# B&R Automation Studio project URTC-with-integrated-CNC-system-main
Automation Studio 4.5.2.102

## Configuration Real

CPU 4PP065.0571-P74, AutomationRuntime D4.52, Build 4.1.2, Vc V4.25.0, Safety 1.6

### Task classes (Cpu.sw)
```
Cyclic#1 (cycle 2000 us, tolerance 0 us):
  ncsdcctrl <- ncsdcctrl.prg
  SDCAxisCtr <- SDCAxisCtr.prg
  SDCAxisCt1 <- SDCAxisCtr1.prg
  SDCAxisCt2 <- SDCAxisCtr2.prg
DataObjects: Arnc0sys
NcDataObjects: AxisInit <- AxisInit.dob, gAxis03a <- gAxis03obj.gAxis03a.dob, gAxis03i <- gAxis03obj.gAxis03i.dob, AxisApt <- AxisApt.dob, gmcipvar <- GmcIpUserConfig.gmcipvar.dob, gmcipfun <- GmcIpUserConfig.gmcipfun.dob, gmcipfub <- GmcIpUserConfig.gmcipfub.dob, gmcipubr <- GmcIpUserConfig.gmcipubr.dob, gmcipusm <- GmcIpUserConfig.gmcipusm.dob, gmcipui <- GmcIpUserConfig.gmcipui.dob, gmcipus <- GmcIpUserConfig.gmcipus.dob, gmcipuc <- GmcIpUserConfig.gmcipuc.dob, gmcipsys <- GmcIpConfig.gmcipsys.dob, gmciplbr <- GmcIpConfig.gmciplbr.dob, gmcipcbr <- GmcIpConfig.gmcipcbr.dob, gmciplsm <- GmcIpConfig.gmciplsm.dob, gmcipcsm <- GmcIpConfig.gmcipcsm.dob, gmcipcfg <- GmcIpConfig.gmcipcfg.dob, gmcipiec <- GmcIpConfig.gmcipiec.dob, gmciplog <- GmcIpConfig.gmciplog.dob, gmcipesm <- GmcIpConfig.gmcipesm.dob, gmcipmxd <- GmcIpConfig.gmcipmxd.dob, gmcipmx <- GmcIpConfig.gmcipmx.dob, CncInit <- CncInit.dob, CncProg <- CncProg.dob, CncProg1 <- CncProg1.dob, gAxis04a <- gAxis04obj.gAxis04a.dob, gAxis04i <- gAxis04obj.gAxis04i.dob
Binaries: TCData, Acp10map1, acp10cfg, Acp10map, arconfig, User, Role, sysconf, iomap, asfw, ashwd, arnc0cfg, Arnc0map
Libraries: Acp10sdc, Library, Acp10man, Acp10_MC, sys_lib, brsystem, asstring, powerlnk, asieccon, AsMath, Arnc0man, DataObj, AsArLog, FileIO, AsArProf, AsMem, Runtime, astime, Acp10par, NcGlobal, asiotime, AsBrStr
```

### Hardware
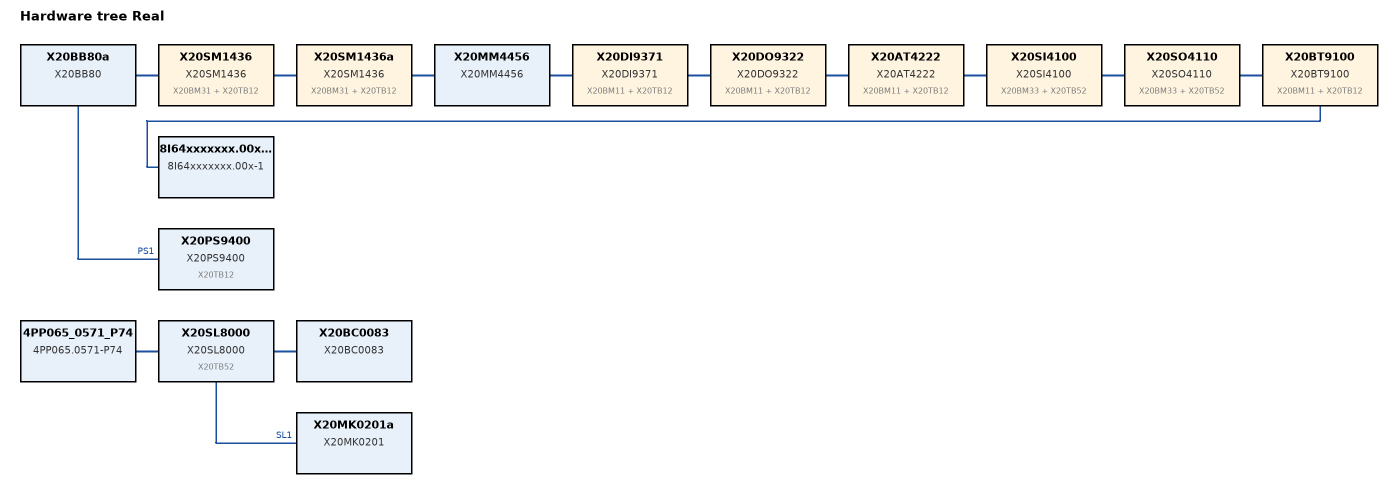
```
4PP065_0571_P74 : 4PP065.0571-P74 v1.1.2.0
  Connector IF4:
    EplInterfaceRedundant = 0
    EplEthInterfaceRedundant = 0
  Connector IF5:
    ActivateDevice = 1
    Mode = Manual
    InternetAddress = 10.0.1.10
    SubnetMask = 255.255.255.0
  ConfigurationID = labBR
  TimerDeviceType = EPLX2X
  TimerDevice = 4PP065_0571_P74.IF4
  TaskClassIdleTime = 2000
  Cyclic1Duration = 2000
  Cyclic1Tolerance = 0
  Cyclic1Output = 1
  Cyclic3Tolerance = 0
  VcObjectName = Visu
8I64xxxxxxx.00x-1 : 8I64xxxxxxx.00x-1 v2.1.2.0  [X2X1 -> X20BT9100.X2X1 [Cable Type=X2XCable, Length=10, Version=1.0.0.2]]
  BothEndSwitchesAreNormallyOpen_r1 = on
  QuickStopIsNormallyOpen_r1 = on
X20AT4222 : X20AT4222 v1.2.3.0  [SS1 -> X20TB12f.SS; SL -> X20BM11c.SL1]
X20BB80a : X20BB80 v1.0.2.0
X20BC0083 : X20BC0083 v2.9.0.0  [PLK1 -> X20SL8000.PLK2 (NodeNumber=2) [Cable Type=PowerlinkCable, Length=10, Version=1.0.0.2]; SL -> X20BB80a.SL1]
X20BM11a : X20BM11 v1.0.0.1  [X2X1 -> X20MM4456.X2X2]
X20BM11b : X20BM11 v1.0.0.1  [X2X1 -> X20BM11a.X2X2]
X20BM11c : X20BM11 v1.0.0.1  [X2X1 -> X20BM11b.X2X2]
X20BM11d : X20BM11 v1.0.0.1  [X2X1 -> X20BM33b.X2X2]
X20BM31a : X20BM31 v1.0.0.1  [X2X1 -> X20BB80a.IF1]
X20BM31b : X20BM31 v1.0.0.1  [X2X1 -> X20BM31a.X2X2]
X20BM33a : X20BM33 v1.0.0.4  [X2X1 -> X20BM11c.X2X2]
X20BM33b : X20BM33 v1.0.0.4  [X2X1 -> X20BM33a.X2X2]
X20BT9100 : X20BT9100 v1.0.3.0  [SS1 -> X20TB12g.SS; SL -> X20BM11d.SL1]
X20DI9371 : X20DI9371 v1.0.2.0  [SS1 -> X20TB12d.SS; SL -> X20BM11a.SL1]
X20DO9322 : X20DO9322 v1.0.3.0  [SS1 -> X20TB12e.SS; SL -> X20BM11b.SL1]
X20MK0201a : X20MK0201 v1.0.0.0  [SL -> X20SL8000.SL1]
X20MM4456 : X20MM4456 v1.1.5.0  [X2X1 -> X20BM31b.X2X2]
X20PS9400 : X20PS9400 v1.0.2.4  [SS1 -> X20TB12b.SS; PS -> X20BB80a.PS1]
X20SI4100 : X20SI4100 v1.10.1.1  [SS1 -> X20TB52b.SS; SL -> X20BM33a.SL1]
X20SL8000 : X20SL8000 v1.6.5.1  [PLK1 -> 4PP065_0571_P74.IF4 (NodeNumber=1) [Cable Type=PowerlinkCable, Length=10, Version=1.0.0.2]; PLK2 -> X20BC0083.PLK1 (NodeNumber=1) [Cable Type=PowerlinkCable, Length=10, Version=1.0.0.2]; SS1 -> X20TB52a.SS]
  SafeProject = SafeLOGIC-1
X20SM1436 : X20SM1436 v1.4.2.1  [SS1 -> X20TB12a.SS; SL -> X20BM31a.SL1]
X20SM1436a : X20SM1436 v1.4.2.1  [SS1 -> X20TB12c.SS; SL -> X20BM31b.SL1]
X20SO4110 : X20SO4110 v1.10.1.1  [SS1 -> X20TB52c.SS; SL -> X20BM33b.SL1]
  SafeLogicID = 2
  SafeModuleID = 3
X20TB12a : X20TB12 v1.0.0.0
X20TB12b : X20TB12 v1.0.0.0
X20TB12c : X20TB12 v1.0.0.0
X20TB12d : X20TB12 v1.0.0.0
X20TB12e : X20TB12 v1.0.0.0
X20TB12f : X20TB12 v1.0.0.0
X20TB12g : X20TB12 v1.0.0.0
X20TB52a : X20TB52 v1.0.0.1
X20TB52b : X20TB52 v1.0.0.1
X20TB52c : X20TB52 v1.0.0.1
```

### Acp10map.ncm - 4PP065_0571_P74/Motion/Acp10map.ncm
```
NcMapping (NcSwId=Acp10, DisabledNodesAreHidden=False)
  NcObject gAxis03 (ModuleId=8I64xxxxxxx.00x-1, ModuleAddress=SDC_IF1.ST1, Type=ncAXIS, Channel=1, AcoposSimulation=Off, InitParameter=gAxis03i, AcoposParameter=gAxis03a, AdditionalData=CNC_Enabled="1" , Disabled=FALSE, ModuleDisabled=FALSE)
```

### Acp10map1.ncm - 4PP065_0571_P74/Motion/Acp10map1.ncm
```
NcMapping (NcSwId=ACP10, DisabledNodesAreHidden=False)
  NcObject AxisX (ModuleAddress=SDC_IF1.ST2, InterfaceType=SDC, Type=ncAXIS, Channel=1, AcoposSimulation=Off, InitParameter=AxisInit, AcoposParameter=AxisApt, AdditionalData=CNC_Enabled="1" , Disabled=FALSE, ModuleDisabled=FALSE)
  NcObject AxisY (ModuleAddress=SDC_IF1.ST3, InterfaceType=SDC, Type=ncAXIS, Channel=1, AcoposSimulation=Off, InitParameter=AxisInit, AcoposParameter=AxisApt, AdditionalData=CNC_Enabled="1" , Disabled=FALSE)
  NcObject AxisZ (ModuleAddress=SDC_IF1.ST4, InterfaceType=SDC, Type=ncAXIS, Channel=1, AcoposSimulation=Off, InitParameter=AxisInit, AcoposParameter=AxisApt, AdditionalData=CNC_Enabled="1" , Disabled=FALSE)
```

### Arnc0map.ncm - 4PP065_0571_P74/Motion/Arnc0map.ncm
```
NcMapping (NcSwId=Arnc0, DisabledNodesAreHidden=False)
  NcObject CNCsys (Type=ncCNCSYS, Channel=1, AcoposSimulation=Off, InitParameter=CncInit, Disabled=FALSE, ModuleDisabled=FALSE)
  NcObject CNC2 (Type=ncCNCSYS, Channel=2, AcoposSimulation=Off, Disabled=TRUE, ModuleDisabled=FALSE)
  NcObject CNC3 (Type=ncCNCSYS, Channel=3, AcoposSimulation=Off, Disabled=TRUE, ModuleDisabled=FALSE)
  NcObject CNC4 (Type=ncCNCSYS, Channel=4, AcoposSimulation=Off, Disabled=TRUE, ModuleDisabled=FALSE)
  NcObject CNC5 (Type=ncCNCSYS, Channel=5, AcoposSimulation=Off, Disabled=TRUE, ModuleDisabled=FALSE)
  NcObject CNC6 (Type=ncCNCSYS, Channel=6, AcoposSimulation=Off, Disabled=TRUE, ModuleDisabled=FALSE)
  NcObject CNC7 (Type=ncCNCSYS, Channel=7, AcoposSimulation=Off, Disabled=TRUE, ModuleDisabled=FALSE)
  NcObject CNC8 (Type=ncCNCSYS, Channel=8, AcoposSimulation=Off, Disabled=TRUE, ModuleDisabled=FALSE)
  NcObject CNC9 (Type=ncCNCSYS, Channel=9, AcoposSimulation=Off, Disabled=TRUE, ModuleDisabled=FALSE)
  NcObject CNC10 (Type=ncCNCSYS, Channel=10, AcoposSimulation=Off, Disabled=TRUE, ModuleDisabled=FALSE)
  NcObject CNC11 (Type=ncCNCSYS, Channel=11, AcoposSimulation=Off, Disabled=TRUE, ModuleDisabled=FALSE)
  NcObject CNC12 (Type=ncCNCSYS, Channel=12, AcoposSimulation=Off, Disabled=TRUE, ModuleDisabled=FALSE)
  NcObject CNC13 (Type=ncCNCSYS, Channel=13, AcoposSimulation=Off, Disabled=TRUE, ModuleDisabled=FALSE)
  NcObject CNC14 (Type=ncCNCSYS, Channel=14, AcoposSimulation=Off, Disabled=TRUE, ModuleDisabled=FALSE)
  NcObject CNC15 (Type=ncCNCSYS, Channel=15, AcoposSimulation=Off, Disabled=TRUE, ModuleDisabled=FALSE)
  NcObject CNC16 (Type=ncCNCSYS, Channel=16, AcoposSimulation=Off, Disabled=TRUE, ModuleDisabled=FALSE)
  NcObject CNC17 (Type=ncCNCSYS, Channel=17, AcoposSimulation=Off, Disabled=TRUE, ModuleDisabled=FALSE)
  NcObject CNC18 (Type=ncCNCSYS, Channel=18, AcoposSimulation=Off, Disabled=TRUE, ModuleDisabled=FALSE)
  NcObject CNC19 (Type=ncCNCSYS, Channel=19, AcoposSimulation=Off, Disabled=TRUE, ModuleDisabled=FALSE)
  NcObject CNC20 (Type=ncCNCSYS, Channel=20, AcoposSimulation=Off, Disabled=TRUE, ModuleDisabled=FALSE)
  NcObject CNC21 (Type=ncCNCSYS, Channel=21, AcoposSimulation=Off, Disabled=TRUE, ModuleDisabled=FALSE)
  NcObject CNC22 (Type=ncCNCSYS, Channel=22, AcoposSimulation=Off, Disabled=TRUE, ModuleDisabled=FALSE)
  NcObject CNC23 (Type=ncCNCSYS, Channel=23, AcoposSimulation=Off, Disabled=TRUE, ModuleDisabled=FALSE)
  NcObject CNC24 (Type=ncCNCSYS, Channel=24, AcoposSimulation=Off, Disabled=TRUE, ModuleDisabled=FALSE)
```

## Logical view

### Global.var - Global variables
```iecst
VAR
	AxisX : ACP10AXIS_typ := (0);
	AxisX_EncIf : SdcEncIf16_typ := (0);
	AxisX_DrvIf : SdcDrvIf16_typ := (0);
	AxisX_DiDoIf : SdcDiDoIf_typ := (0);
	AxisX_HW : SdcHwCfg_typ := (0);
	AxisY : ACP10AXIS_typ := (0);
	AxisY_EncIf : SdcEncIf16_typ := (0);
	AxisY_DrvIf : SdcDrvIf16_typ := (0);
	AxisY_DiDoIf : SdcDiDoIf_typ := (0);
	AxisY_HW : SdcHwCfg_typ := (0);
	AxisZ : ACP10AXIS_typ := (0);
	AxisZ_EncIf : SdcEncIf16_typ := (0);
	AxisZ_DrvIf : SdcDrvIf16_typ := (0);
	AxisZ_DiDoIf : SdcDiDoIf_typ := (0);
	AxisZ_HW : SdcHwCfg_typ := (0);
	gAxis01 : ACP10AXIS_typ := (0);
	gAxis02 : ACP10AXIS_typ := (0);
	gAxisTest : ACP10AXIS_typ := (0);
	gAxisTest_HW : SdcHwCfg_typ := (0);
	gAxisTest_DrvIf : SdcDrvIf16_typ := (0);
	gAxisTest_DiDoIf : SdcDiDoIf_typ := (0);
	gAxisTest_ModuleOk : BOOL := 0;
	gAxis03 : ACP10AXIS_typ := (0);
	gAxis03_HW : SdcHwCfg_typ := (0);
	gAxis03_DrvIf : SdcDrvIf16_typ := (0);
	gAxis03_DiDoIf : SdcDiDoIf_typ := (0);
	gAxis03_ModuleOk : BOOL := 0;
	CNCsys : ARNC0CNC_typ;
	position : INT := 0;
	Myspeed : INT := 0;
	gAxis04 : ACP10AXIS_typ := (0);
	gAxis04_HW : SdcHwCfg_typ := (0);
	gAxis04_DrvIf : SdcDrvIf16_typ := (0);
	gAxis04_EncIf1 : SdcEncIf16_typ := (0);
	gAxis04_DiDoIf : SdcDiDoIf_typ := (0);
	gAxis04_MotorStep0 : INT := 0;
END_VAR
```

### Data object Logical/AxisInit (Ax)

#### AxInitAcp10.ax
```
InitParameter (Version=3.13.1, NcSwId=ACP10)
  ACP10AXIS_typ:
    dig_in:
      level:
        reference = ncACTIV_HI
        pos_hw_end = ncACTIV_HI
        neg_hw_end = ncACTIV_HI
        trigger1 = ncACTIV_HI
        trigger2 = ncACTIV_HI
    encoder_if:
      parameter:
        count_dir = ncSTANDARD
        scaling:
          load:
            units = 3000
            rev_motor = 1
    limit:
      parameter:
        v_pos = 7500.0
        v_neg = 7500.0
        a1_pos = 10000.0
        a2_pos = 10000.0
        a1_neg = 10000.0
        a2_neg = 10000.0
        t_jolt = 0.0
        t_in_pos = 0.0
        pos_sw_end = 8388607
        neg_sw_end = -8388608
        ds_warning = 500.0
        ds_stop = 10000.0
        a_stop = 1.0E+30
        dv_stop = 0.0
        dv_stop_mode = ncOFF
    controller:
      mode = ncPOSITION
      position:
        kv = 10.0
        tn = 0.0
        t_predict = 0.04
        t_total = 0.04
        p_max = 10000.0
        i_max = 0.0
      speed:
        kv = 2.0
        tn = 0.0
        t_filter = 0.0
        isq_filter1:
          type = ncOFF
          a0 = 0.0
          a1 = 0.0
          b0 = 0.0
          b1 = 0.0
          b2 = 0.0
          c0_par_id = 0
          c1_par_id = 0
        isq_filter2:
          type = ncOFF
          a0 = 0.0
          a1 = 0.0
          b0 = 0.0
          b1 = 0.0
          b2 = 0.0
          c0_par_id = 0
          c1_par_id = 0
        isq_filter3:
          type = ncOFF
          a0 = 0.0
          a1 = 0.0
          b0 = 0.0
          b1 = 0.0
          b2 = 0.0
          c0_par_id = 0
          c1_par_id = 0
      uf:
        type = ncLINEAR
        auto_config = ncMOTOR_PAR
        u0 = 0.0
        un = 0.0
        fn = 50.0
        k_f_slip = 0.0
      ff:
        torque_load = 0.0
        torque_pos = 0.0
        torque_neg = 0.0
        kv_torque = 0.0
        inertia = 0.0
        t_filter_a = 0.0
    move:
      stop:
        parameter[0]:
          decel_ramp = ncA_LIMIT
          controller = ncON
        parameter[1]:
          decel_ramp = ncA_LIMIT
          controller = ncON
        parameter[2]:
          decel_ramp = ncA_LIMIT
          controller = ncON
        parameter[3]:
          decel_ramp = ncA_LIMIT
          controller = ncON
        quickstop:
          decel_ramp = ncA_LIMIT
        drive_error:
          decel_ramp = ncA_LIMIT
      homing:
        parameter:
          s = 0
          v_switch = 6000.0
          v_trigger = 2000.0
          a = 10000.0
          mode = ncDIRECT
          edge_sw = ncNEGATIVE
          start_dir = ncPOSITIVE
          trigg_dir = ncNEGATIVE
          ref_pulse = ncOFF
          fix_dir = ncOFF
          tr_s_block = 0.0
          torque_lim = 0.0
          ds_block = 0.0
          ds_stop = 0.0
      basis:
        parameter:
          v_pos = 4000.0
          v_neg = 4000.0
          a1_pos = 10000.0
          a2_pos = 10000.0
          a1_neg = 10000.0
          a2_neg = 10000.0
    message:
      text:
        parameter:
          format = ncBREAK
          columns = 80
          data_modul
```

### Program Logical/ncsdcctrl (IEC)

#### ncsdcctrl.var
```iecst
VAR
	gAxis04_oSetPosOld : INT := 0;
END_VAR
```

#### ncsdcctrlCyclic.st
```iecst
PROGRAM _CYCLIC

(* ### BEGIN gAxisTest ### *)

(* life counter emulation of digital inputs *)
 gAxisTest_DiDoIf.iLifeCntReference := gAxisTest_DiDoIf.iLifeCntReference + 1;
 gAxisTest_DiDoIf.iLifeCntNegHwEnd  := gAxisTest_DiDoIf.iLifeCntNegHwEnd  + 1;
 gAxisTest_DiDoIf.iLifeCntPosHwEnd  := gAxisTest_DiDoIf.iLifeCntPosHwEnd  + 1;

(* ### END gAxisTest ### *)

(* ### BEGIN gAxis03 ### *)

(* life counter emulation of digital inputs *)
 gAxis03_DiDoIf.iLifeCntReference := gAxis03_DiDoIf.iLifeCntReference + 1;
 gAxis03_DiDoIf.iLifeCntNegHwEnd  := gAxis03_DiDoIf.iLifeCntNegHwEnd  + 1;
 gAxis03_DiDoIf.iLifeCntPosHwEnd  := gAxis03_DiDoIf.iLifeCntPosHwEnd  + 1;

(* ### END gAxis03 ### *)

(* ### BEGIN gAxis04 ### *)

(* life counter emulation of digital inputs *)
       gAxis04_DiDoIf.iLifeCntReference := gAxis04_DiDoIf.iLifeCntReference + 1;
       gAxis04_DiDoIf.iLifeCntNegHwEnd  := gAxis04_DiDoIf.iLifeCntNegHwEnd  + 1;
       gAxis04_DiDoIf.iLifeCntPosHwEnd  := gAxis04_DiDoIf.iLifeCntPosHwEnd  + 1;

(* default function model of ACOPOSmicro: convert absolute steps to delta steps - overflow save delta calculation *)
       gAxis04_MotorStep0 := gAxis04_DrvIf.oSetPos - gAxis04_oSetPosOld;
       gAxis04_oSetPosOld := gAxis04_DrvIf.oSetPos;

(* ### END gAxis04 ### *)

END_PROGRAM
```

#### ncsdcctrlInit.st
```iecst
PROGRAM _INIT

(* ### BEGIN gAxisTest ### *)

(* initialize variables *)
 gAxisTest_HW.DrvIf_Typ := ncSDC_DRVSERVO16;
 strcpy( ADR(gAxisTest_HW.DrvIf_Name[0]), ADR('gAxisTest_DrvIf') );
 gAxisTest_HW.DiDoIf_Typ := ncSDC_DIDO;
 strcpy( ADR(gAxisTest_HW.DiDoIf_Name[0]), ADR('gAxisTest_DiDoIf') );

(* force variable offset generation *)
 gAxisTest.size                      := gAxisTest.size;
 gAxisTest_DrvIf.iLifeCnt            := gAxisTest_DrvIf.iLifeCnt;
 gAxisTest_DiDoIf.iLifeCntDriveReady := gAxisTest_DiDoIf.iLifeCntDriveReady;
 gAxisTest_ModuleOk                  := gAxisTest_ModuleOk;

(* assign your hardware inputs here*)

(* gAxisTest_DiDoIf.iPosHwEnd  := gAxisTest_DiDoIf.iPosHwEnd;
 gAxisTest_DiDoIf.iNegHwEnd  := gAxisTest_DiDoIf.iNegHwEnd;
 gAxisTest_DiDoIf.iReference := gAxisTest_DiDoIf.iReference;
 *)

(* ### END gAxisTest ### *)

(* ### BEGIN gAxis03 ### *)

(* initialize variables *)
 gAxis03_HW.DrvIf_Typ := ncSDC_DRVSERVO16;
 strcpy( ADR(gAxis03_HW.DrvIf_Name[0]), ADR('gAxis03_DrvIf') );
 gAxis03_HW.DiDoIf_Typ := ncSDC_DIDO;
 strcpy( ADR(gAxis03_HW.DiDoIf_Name[0]), ADR('gAxis03_DiDoIf') );

(* force variable offset generation *)
 gAxis03.size                      := gAxis03.size;
 gAxis03_DrvIf.iLifeCnt            := gAxis03_DrvIf.iLifeCnt;
 gAxis03_DiDoIf.iLifeCntDriveReady := gAxis03_DiDoIf.iLifeCntDriveReady;
 gAxis03_ModuleOk                  := gAxis03_ModuleOk;

(* assign your hardware inputs here*)

(* gAxis03_DiDoIf.iPosHwEnd  := gAxis03_DiDoIf.iPosHwEnd;
 gAxis03_DiDoIf.iNegHwEnd  := gAxis03_DiDoIf.iNegHwEnd;
 gAxis03_DiDoIf.iReference := gAxis03_DiDoIf.iReference;
 *)

(* ### END gAxis03 ### *)

(* ### BEGIN gAxis04 ### *)

(* initialize general interfaces *)
       gAxis04.size := gAxis04.size;
       gAxis04_HW.DrvIf_Typ := ncSDC_DRVSM16;
       brsstrcpy( ADR(gAxis04_HW.DrvIf_Name[0]), ADR('gAxis04_DrvIf') );
       gAxis04_HW.DiDoIf_Typ := ncSDC_DIDO;
       brsstrcpy( ADR(gAxis04_HW.DiDoIf_Name[0]), ADR('gAxis04_DiDoIf') );
       gAxis04_HW.EncIf1_Typ := ncSDC_ENC16;
       brsstrcpy( ADR(gAxis04_HW.EncIf1_Name[0]), ADR('gAxis04_EncIf1') );
       gAxis04_EncIf1.iLifeCnt := gAxis04_EncIf1.iLifeCnt;

(* initialize old-value for delta step calculation *)
       gAxis04_oSetPosOld := gAxis04_DrvIf.oSetPos;

(* ### END gAxis04 ### *)

END_PROGRAM
```

### Data object Logical/CncInit (Cns)

- CncInit.cns (not shown)

### Data object Logical/CncProg (Cnc)

#### CncProg.cnc
```
%001 (CncProgram)
N10 G01 X0 Z1000 F300000
N20 G01 X0 Z3000 F360000
N20 M30
```

### Program Logical/SDCAxisCtr (ANSIC)

#### Variables.var
```iecst
VAR
	axis_X : FB_Axis;
	coil_powered : BOOL := FALSE;
	coil_pwm_value : {REDUND_UNREPLICABLE} INT := 200;
	desired_speed : INT := 0;
	fb_controller : FB_Controller;
	min_task : INT := 7000;
	pwm_period : {REDUND_UNREPLICABLE} UINT := 200;
	lagerror : USINT := 0;
END_VAR
```

#### Main.c
```c
#include <bur/plctypes.h>

#ifdef _DEFAULT_INCLUDES
	#include <AsDefault.h>
#endif

void increase_counters(void);

void _INIT ProgramInit(void)
{
	//Устанваливаем типы SDC модулей
	AxisX_HW.EncIf1_Typ = ncSDC_ENC16;
	AxisX_HW.DiDoIf_Typ = ncSDC_DIDO;
	AxisX_HW.DrvIf_Typ = ncSDC_DRVSERVO16;

	//Устанавливаем имена переменных
	strcpy(AxisX_HW.EncIf1_Name, "AxisX_EncIf");
	strcpy(AxisX_HW.DrvIf_Name, "AxisX_DrvIf");
	strcpy(AxisX_HW.DiDoIf_Name, "AxisX_DiDoIf");

	//Устанавливаем входы готовности и нормальной работы
	AxisX_EncIf.iEncOK = 1;
	AxisX_DrvIf.iDrvOK = 1;
	AxisX_DrvIf.iStatusEnable = 1;
	AxisX_DiDoIf.iDriveReady = 1;

	fb_controller.dt = 0.002;
	fb_controller.k_i = 0.16;
	fb_controller.k_p = 0.0064;
	fb_controller.max_abs_value = 24.0;

	pwm_period = 200;
}

void _CYCLIC ProgramCyclic(void)
{
	position = AxisX.monitor.s;
	Myspeed = AxisX.monitor.v;
	FB_Axis(&axis_X);
	coil_pwm_value = coil_powered ? 32767 : 0;

	increase_counters();

	//Формирование показаний датчика

	AxisX_EncIf.iActTime = (INT)	AsIOTimeCyclicStart();
	AxisX_EncIf.iActPos = axis_X.counter;
	AxisX_DiDoIf.iPosHwEnd = axis_X.endswitch_a_reached;
	AxisX_DiDoIf.iNegHwEnd = axis_X.endswitch_b_reached;
	fb_controller.in = AxisX_DrvIf.oSetPos;

	if((fb_controller.in<min_task)&&(fb_controller.in>(-min_task))) fb_controller.in = 0;
	fb_controller.in = fb_controller.in * 6500/32767 - axis_X.speed;

	FB_Controller(&fb_controller);

	axis_X.pwm_value = fb_controller.out / 24.0 * 32767;
}

void increase_counters(void)
{
	AxisX_EncIf.iLifeCnt++;
	AxisX_DiDoIf.iLifeCntDriveEnable++;
	AxisX_DiDoIf.iLifeCntDriveReady++;
	AxisX_DiDoIf.iLifeCntNegHwEnd++;
	AxisX_DiDoIf.iLifeCntPosHwEnd++;
	AxisX_DiDoIf.iLifeCntReference++;
	AxisX_DrvIf.iLifeCnt++;
}

void _EXIT ProgramExit(void)
{
	// Insert code here

}
```

### Program Logical/SDCAxisCtr1 (ANSIC)

#### Main.c
```c
#include <bur/plctypes.h>

#ifdef _DEFAULT_INCLUDES
	#include <AsDefault.h>
#endif

void increase_counters(void);

void _INIT ProgramInit(void)
{
	//Устанваливаем типы SDC модулей
	//Устанваливаем типы SDC модулей
	AxisY_HW.EncIf1_Typ = ncSDC_ENC16;
	AxisY_HW.DiDoIf_Typ = ncSDC_DIDO;
	AxisY_HW.DrvIf_Typ = ncSDC_DRVSERVO16;

	//Устанавливаем имена переменных
	strcpy(AxisY_HW.EncIf1_Name, "AxisY_EncIf");
	strcpy(AxisY_HW.DrvIf_Name, "AxisY_DrvIf");
	strcpy(AxisY_HW.DiDoIf_Name, "AxisY_DiDoIf");

	//Устанавливаем входы готовности и нормальной работы
	AxisY_EncIf.iEncOK = 1;
	AxisY_DrvIf.iDrvOK = 1;
	AxisY_DrvIf.iStatusEnable = 1;
	AxisY_DiDoIf.iDriveReady = 1;

	fb_controller.dt = 0.002;
	fb_controller.k_i = 0.16;
	fb_controller.k_p = 0.0064;
	fb_controller.max_abs_value = 24.0;

	pwm_period = 200;

	//Устанавливаем имена переменных

	//Устанавливаем входы готовности и нормальной работы

}

void _CYCLIC ProgramCyclic(void)
{

	FB_Axis(&axis_Y);
	coil_pwm_value = coil_powered ? 32767 : 0;

	increase_counters();

	//Формирование показаний датчика

	AxisY_EncIf.iActTime = (INT)	AsIOTimeCyclicStart();
	AxisY_EncIf.iActPos = axis_Y.counter;
	AxisY_DiDoIf.iPosHwEnd = axis_Y.endswitch_b_reached;
	AxisY_DiDoIf.iNegHwEnd = axis_Y.endswitch_a_reached;
	fb_controller.in = AxisY_DrvIf.oSetPos;

	if((fb_controller.in<min_task)&&(fb_controller.in>(-min_task))) fb_controller.in = 0;
	fb_controller.in = fb_controller.in * 6500/32767 - axis_Y.speed;

	FB_Controller(&fb_controller);

	axis_Y.pwm_value = fb_controller.out / 24.0 * 32767;
	//Формирование показаний датчика

}

void increase_counters(void)
{

		AxisY_EncIf.iLifeCnt++;
		AxisY_DiDoIf.iLifeCntDriveEnable++;
		AxisY_DiDoIf.iLifeCntDriveReady++;
		AxisY_DiDoIf.iLifeCntNegHwEnd++;
		AxisY_DiDoIf.iLifeCntPosHwEnd++;
		AxisY_DiDoIf.iLifeCntReference++;
		AxisY_DrvIf.iLifeCnt++;

}

void _EXIT ProgramExit(void)
{
	// Insert code here

}
```

### Program Logical/SDCAxisCtr2 (ANSIC)

#### Main.c
```c
#include <bur/plctypes.h>

#ifdef _DEFAULT_INCLUDES
	#include <AsDefault.h>
#endif

void increase_counters(void);

void _INIT ProgramInit(void)
{
	//Устанваливаем типы SDC модулей

	//Устанваливаем типы SDC модулей
	AxisZ_HW.EncIf1_Typ = ncSDC_ENC16;
	AxisZ_HW.DiDoIf_Typ = ncSDC_DIDO;
	AxisZ_HW.DrvIf_Typ = ncSDC_DRVSERVO16;

	//Устанавливаем имена переменных
	strcpy(AxisZ_HW.EncIf1_Name, "AxisZ_EncIf");
	strcpy(AxisZ_HW.DrvIf_Name, "AxisZ_DrvIf");
	strcpy(AxisZ_HW.DiDoIf_Name, "AxisZ_DiDoIf");

	//Устанавливаем входы готовности и нормальной работы
	AxisZ_EncIf.iEncOK = 1;
	AxisZ_DrvIf.iDrvOK = 1;
	AxisZ_DrvIf.iStatusEnable = 1;
	AxisZ_DiDoIf.iDriveReady = 1;

	fb_controller.dt = 0.002;
	fb_controller.k_i = 0.16;
	fb_controller.k_p = 0.0064;
	fb_controller.max_abs_value = 24.0;

	pwm_period = 200;
	//Устанавливаем имена переменных

	//Устанавливаем входы готовности и нормальной работы

}

void _CYCLIC ProgramCyclic(void)
{
	FB_Axis(&axis_Z);
	coil_pwm_value = coil_powered ? 32767 : 0;

	increase_counters();

	//Формирование показаний датчика

	AxisZ_EncIf.iActTime = (INT)	AsIOTimeCyclicStart();
	AxisZ_EncIf.iActPos = axis_Z.counter;
	AxisZ_DiDoIf.iPosHwEnd = axis_Z.endswitch_a_reached;
	AxisZ_DiDoIf.iNegHwEnd = axis_Z.endswitch_b_reached;
	fb_controller.in = AxisZ_DrvIf.oSetPos;

	if((fb_controller.in<min_task)&&(fb_controller.in>(-min_task))) fb_controller.in = 0;
	fb_controller.in = fb_controller.in * 6500/32767 - axis_Z.speed;

	FB_Controller(&fb_controller);

	axis_Z.pwm_value = fb_controller.out / 24.0 * 32767;

}

void increase_counters(void)
{
	AxisZ_EncIf.iLifeCnt++;
	AxisZ_DiDoIf.iLifeCntDriveEnable++;
	AxisZ_DiDoIf.iLifeCntDriveReady++;
	AxisZ_DiDoIf.iLifeCntNegHwEnd++;
	AxisZ_DiDoIf.iLifeCntPosHwEnd++;
	AxisZ_DiDoIf.iLifeCntReference++;
	AxisZ_DrvIf.iLifeCnt++;
}

void _EXIT ProgramExit(void)
{
	// Insert code here

}
```

### Data object Logical/CncProg1 (Cnc)

#### CncProg.cnc
```
%001 (CncProgram)

N10 G01 Z1000 F300000
N20 G01 Z3000 F360000
N20 M30
```

### Package Logical/gAxis04obj - gAxis04obj

### gAxis04i.ax
```
InitParameter (Version=3.13.1, NcSwId=Acp10)
  ACP10AXIS_typ:
    dig_in:
      level:
        reference = ncACTIV_HI
        pos_hw_end = ncACTIV_LO
        neg_hw_end = ncACTIV_LO
        trigger1 = ncACTIV_HI
        trigger2 = ncACTIV_LO + ncQUICKSTOP
    encoder_if:
      parameter:
        count_dir = ncSTANDARD
        scaling:
          load:
            units = 1000
            rev_motor = 1
    limit:
      parameter:
        v_pos = 10000
        v_neg = 10000
        a1_pos = 50000
        a2_pos = 50000
        a1_neg = 50000
        a2_neg = 50000
        t_jolt = 0
        t_in_pos = 0
        pos_sw_end = 2000000000
        neg_sw_end = -2000000000
        ds_warning = 500
        ds_stop = 1000
        a_stop = 1.0e30
        dv_stop = 0
        dv_stop_mode = ncOFF
    controller:
      mode = ncPOSITION
      position:
        kv = 50
        tn = 0
        t_predict = 0.01
        t_total = 0.01
        p_max = 1.0e30
        i_max = 0
      speed:
        kv = 2.0
        tn = 0
        t_filter = 0.0
        isq_filter1:
          type = ncOFF
          a0 = 0.0
          a1 = 0.0
          b0 = 0.0
          b1 = 0.0
          b2 = 0.0
          c0_par_id = 0
          c1_par_id = 0
        isq_filter2:
          type = ncOFF
          a0 = 0.0
          a1 = 0.0
          b0 = 0.0
          b1 = 0.0
          b2 = 0.0
          c0_par_id = 0
          c1_par_id = 0
        isq_filter3:
          type = ncOFF
          a0 = 0.0
          a1 = 0.0
          b0 = 0.0
          b1 = 0.0
          b2 = 0.0
          c0_par_id = 0
          c1_par_id = 0
      uf:
        type = ncLINEAR
        auto_config = ncMOTOR_PAR
        u0 = 0
        un = 0
        fn = 50.0
        k_f_slip = 0
      ff:
        torque_load = 0.0
        torque_pos = 0.0
        torque_neg = 0.0
        kv_torque = 0.0
        inertia = 0.0
        t_filter_a = 0.0
    move:
      stop:
        parameter[0]:
          decel_ramp = ncA_LIMIT
          controller = ncON
        parameter[1]:
          decel_ramp = ncA_LIMIT
          controller = ncON
        parameter[2]:
          decel_ramp = ncA_LIMIT
          controller = ncON
        parameter[3]:
          decel_ramp = ncA_LIMIT
          controller = ncON
        quickstop:
          decel_ramp = ncA_LIMIT
        drive_error:
          decel_ramp = ncA_LIMIT
      homing:
        parameter:
          s = 0
          v_switch = 5000
          v_trigger = 500
          a = 50000
          mode = ncDIRECT
          edge_sw = ncPOSITIVE
          start_dir = ncPOSITIVE
          trigg_dir = ncPOSITIVE
          ref_pulse = ncOFF
          fix_dir = ncOFF
          tr_s_block = 0
          torque_lim = 0
          ds_block = 0
          ds_stop = 0
      basis:
        parameter:
          v_pos = 5000
          v_neg = 5000
          a1_pos = 50000
          a2_pos = 50000
          a1_neg = 50000
          a2_neg = 50000
    message:
      text:
        parameter:
          format = ncBREAK
          columns = 80
          data_modul = acp10etxen
```

Listed in the project but not available here: Logical/Global.typ, Logical/Libraries, Logical/AxisApt, Logical/Types.typ, Logical/acp10etxen, Logical/gAxis03obj, Logical/GmcIpConfig, Logical/GmcIpUserConfig
